{attribute 'qualified_only'}
VAR_GLOBAL
END_VAR

(* stored: Version 1.1.0.1, ProductVersion 3.1.4022.7
   GVL GVL_02_Parameter_Servo_Motor_Shelf_Y: Id {081a547d-4278-4c6b-a502-c00073f9bfc7} *)
